# EPICS substitutions: CARSApp/Db/Pelco_CM6700.substitutions
# Takes macros P, R, PORT
file "$(IP)/db/Pelco_CM6700.db"
{}

file "$(IP)/db/Pelco_CM6700_names.db"
{
pattern
{STR}
{ZRST}
{ONST}
{TWST}
{THST}
{FRST}
{FVST}
{SXST}
{SVST}
{EIST}
{NIST}
{TEST}
{ELST}
{TVST}
{TTST}
{FTST}
{FFST}
}
